{attribute 'qualified_only'}
{attribute 'strict'}
TYPE E_CRYO_CRYOTELGT_STATE :
(
	OFF := 0,
	STARTING,
	ON,
	STOPPING,
	ERROR
);
END_TYPE

(* stored: Version 1.1.0.1, ProductVersion 3.1.4024.12
   DUT E_CRYO_CRYOTELGT_STATE: Id {6def3638-1569-4541-921f-4e2aacb91c19} *)
